{attribute 'linkalways'} 
{attribute 'no_explicit_call' := 'This FB is a CLASS and must be accessed using methods or properties'}
{attribute 'enable_dynamic_creation'}
FUNCTION_BLOCK ContentHost IMPLEMENTS I_Contents, I_Serializable
VAR
	hostParent : I_HostContent;
	eventTarget : I_EventTarget;
	contents : Dictionary;
	selfCreatedContent : Stack;
END_VAR

METHOD PUBLIC Accept
VAR_INPUT
	visitor : I_ContentVisitor;
END_VAR
VAR
	enumerator : I_ForwardEnumerator;
	content : I_Content;
END_VAR
enumerator := contents.GetEnumerator();

WHILE (enumerator.MoveNext()) DO
	
	IF enumerator.TryGet(content) THEN
		content.Accept(Visitor);
	END_IF

END_WHILE

enumerator.Dispose();
END_METHOD

METHOD PUBLIC AddContent
VAR_INPUT
	Content : I_Content;
END_VAR
contents.AddOrUpdate(Content.Name, Content);
EmitOnContentAddedEvent(Content);
END_METHOD

METHOD PUBLIC AddDataAsContent : I_Content
VAR_INPUT
	Name : T_MAXSTRING;
	Data : I_Datatype;
END_VAR
VAR
	content : I_Content;
END_VAR
content := CreateContent(Name, Data);
selfCreatedContent.Push(content);
AddDataAsContent := content;
END_METHOD

METHOD PRIVATE CreateContent : I_Content
VAR_INPUT
	ContentName : T_MAXSTRING;
	ContentData : I_Datatype;
END_VAR
VAR
	pContent : POINTER TO Content;
END_VAR
pContent := __NEW(Content(Name := ContentName, Data := ContentData, Parent := hostParent));
CreateContent := pContent^;
END_METHOD

METHOD PRIVATE DisposeSelfCreatedContent : BOOL
VAR
	content : I_Content;
END_VAR
WHILE selfCreatedContent.TryPop(content) DO
	content.Dispose();
END_WHILE
END_METHOD

METHOD PROTECTED EmitOnContentAddedEvent
VAR_INPUT
	Content : I_Content;
END_VAR
VAR
	pContentAddedEvent : POINTER TO ContentAddedEvent;
END_VAR
IF eventTarget = 0 THEN
	RETURN;
END_IF

pContentAddedEvent := __NEW(ContentAddedEvent(Target := Content));
eventTarget.Emit('OnContentAdded',pContentAddedEvent^);
pContentAddedEvent^.Dispose();
END_METHOD

METHOD FB_exit : BOOL
VAR_INPUT
	bInCopyCode : BOOL; // if TRUE, the exit method is called for exiting an instance that is copied afterwards (online change).
END_VAR
IF bInCopyCode THEN
	RETURN;
END_IF

DisposeSelfCreatedContent();
END_METHOD

METHOD FB_init : BOOL
VAR_INPUT
	bInitRetains : BOOL; // if TRUE, the retain variables are initialized (warm start / cold start)
	bInCopyCode : BOOL;  // if TRUE, the instance afterwards gets moved into the copy code (online change)
	Parent : I_HostContent;
	ParentEventTarget : I_EventTarget;
END_VAR
hostParent := Parent;
eventTarget := parentEventTarget;
END_METHOD

METHOD PUBLIC SerializeWith
VAR_INPUT
	Serializer : I_Serializer;
END_VAR
VAR
	enumerator : I_ForwardEnumerator;
	content : I_Content;
END_VAR
IF contents.Count = 0 THEN
	RETURN;
END_IF

Serializer.AddKey('contents');
Serializer.StartArray();

enumerator := contents.GetEnumerator();

WHILE enumerator.MoveNext() DO
	IF enumerator.TryGet(content) THEN
		content.SerializeWith(Serializer);
	END_IF
END_WHILE

Serializer.EndArray();
enumerator.Dispose();
END_METHOD

METHOD PUBLIC TryGetContentByName : BOOL
VAR_INPUT
	Name : T_MAXSTRING;
	Destination : REFERENCE TO I_Content;
END_VAR
VAR
	content : I_Content;
END_VAR
IF NOT contents.TryGetValue(Name, content) THEN
	RETURN;
END_IF

Destination := content;
TryGetContentByName := TRUE;
END_METHOD

END_FUNCTION_BLOCK

(* stored: Version 1.1.0.1, ProductVersion 3.1.4024.12
   POU ContentHost: Id {f669076c-98b4-4a80-95e6-218c34075d57}, SpecialFunc None
   Folder Constructor: Id {f008522b-915a-458b-a34e-a4b0e3dc9ab0}
   Folder Destructor: Id {00e7ca70-7dfc-4dff-995d-0093bd5ee8e6}
   Folder Private: Id {23a79408-daaa-4d15-91ac-6dc86697ba28}
   Folder Protected: Id {620723ea-20f7-482a-8167-dd0825e3806d}
   Method Accept: Id {a1606e8f-5876-48c0-98f6-46743768f294}
   Method AddContent: Id {1e42df45-60ad-4745-9e46-6fb3980191cc}
   Method AddDataAsContent: Id {58b8f25f-0c66-4286-abf4-d1fab45146a1}
   Method CreateContent: Id {46250da3-e89e-409d-ac35-273b0dbb0c12}
   Method DisposeSelfCreatedContent: Id {032c088f-b9ac-4503-a0f4-bdfa212e7d69}
   Method EmitOnContentAddedEvent: Id {f5818c89-d124-4fae-89ec-6a573e586bff}
   Method FB_exit: Id {26c6e675-826b-462f-aea9-8fc06a71ab1a}
   Method FB_init: Id {e3eea328-9f65-424f-996f-3f82903e3715}
   Method SerializeWith: Id {e6b63081-e905-4fe8-a595-01f60b980081}
   Method TryGetContentByName: Id {076edd3f-d171-46dc-b5e5-26dd2689e196} *)
